FUNCTION TryConvert_LWORD_TO_DATE : BOOL
VAR_INPUT
	in : LWORD;
	out : REFERENCE TO DATE;
END_VAR

IF in > DatatypeLimits.MAX_VALUE_OF_LWORD_WHICH_CAN_BE_HELD_IN_A_DATE THEN
	RETURN;
END_IF

out := LWORD_TO_DATE(in);
TryConvert_LWORD_TO_DATE := TRUE;

END_FUNCTION

(* stored: Version 1.1.0.1, ProductVersion 3.1.4024.12
   POU TryConvert_LWORD_TO_DATE: Id {cdb14e6f-7c02-4dde-aed4-d2dd198ab415}, SpecialFunc None *)
